(* IEC 61131-3 sources: mect_apps/Examples/Allarme_TPAC1007_04_AC/plc, 3 files *)

(* ---- Crosstable.gvl ---- *)
VAR_GLOBAL
	SetPoint_temp AT %QD0.4:REAL;
	Start AT %IX0.8.0:BOOL;
	Average_AnInp1 AT %QD0.776:REAL;
	Alarm_temp AT %IX0.780.0:BOOL;	(* Temperature alarm - Analog input 1 *)
	RTU0_TYPE_PORT AT %ID0.20000:UDINT;
	RTU0_BAUDRATE AT %ID0.20004:UDINT;
	RTU0_STATUS AT %ID0.20008:UDINT;
	RTU0_READS AT %ID0.20012:UDINT;
	RTU0_WRITES AT %ID0.20016:UDINT;
	RTU0_TIMEOUTS AT %ID0.20020:UDINT;
	RTU0_COMM_ERRORS AT %ID0.20024:UDINT;
	RTU0_LAST_ERROR AT %ID0.20028:UDINT;
	RTU0_WRITE_QUEUE AT %ID0.20032:UDINT;
	RTU0_READ_QUEUE AT %ID0.20036:UDINT;
	RTU1_TYPE_PORT AT %ID0.20040:UDINT;
	RTU1_BAUDRATE AT %ID0.20044:UDINT;
	RTU1_STATUS AT %ID0.20048:UDINT;
	RTU1_READS AT %ID0.20052:UDINT;
	RTU1_WRITES AT %ID0.20056:UDINT;
	RTU1_TIMEOUTS AT %ID0.20060:UDINT;
	RTU1_COMM_ERRORS AT %ID0.20064:UDINT;
	RTU1_LAST_ERROR AT %ID0.20068:UDINT;
	RTU1_WRITE_QUEUE AT %ID0.20072:UDINT;
	RTU1_READ_QUEUE AT %ID0.20076:UDINT;
	RTU3_TYPE_PORT AT %ID0.20080:UDINT;
	RTU3_BAUDRATE AT %ID0.20084:UDINT;
	RTU3_STATUS AT %ID0.20088:UDINT;
	RTU3_READS AT %ID0.20092:UDINT;
	RTU3_WRITES AT %ID0.20096:UDINT;
	RTU3_TIMEOUTS AT %ID0.20100:UDINT;
	RTU3_COMM_ERRORS AT %ID0.20104:UDINT;
	RTU3_LAST_ERROR AT %ID0.20108:UDINT;
	RTU3_WRITE_QUEUE AT %ID0.20112:UDINT;
	RTU3_READ_QUEUE AT %ID0.20116:UDINT;
	CAN0_TYPE_PORT AT %ID0.20120:UDINT;
	CAN0_BAUDRATE AT %ID0.20124:UDINT;
	CAN0_STATUS AT %ID0.20128:UDINT;
	CAN0_READS AT %ID0.20132:UDINT;
	CAN0_WRITES AT %ID0.20136:UDINT;
	CAN0_TIMEOUTS AT %ID0.20140:UDINT;
	CAN0_COMM_ERRORS AT %ID0.20144:UDINT;
	CAN0_LAST_ERROR AT %ID0.20148:UDINT;
	CAN0_WRITE_QUEUE AT %ID0.20152:UDINT;
	CAN0_READ_QUEUE AT %ID0.20156:UDINT;
	CAN1_TYPE_PORT AT %ID0.20160:UDINT;
	CAN1_BAUDRATE AT %ID0.20164:UDINT;
	CAN1_STATUS AT %ID0.20168:UDINT;
	CAN1_READS AT %ID0.20172:UDINT;
	CAN1_WRITES AT %ID0.20176:UDINT;
	CAN1_TIMEOUTS AT %ID0.20180:UDINT;
	CAN1_COMM_ERRORS AT %ID0.20184:UDINT;
	CAN1_LAST_ERROR AT %ID0.20188:UDINT;
	CAN1_WRITE_QUEUE AT %ID0.20192:UDINT;
	CAN1_READ_QUEUE AT %ID0.20196:UDINT;
	TCPS_TYPE_PORT AT %ID0.20200:UDINT;
	TCPS_IP_ADDRESS AT %ID0.20204:UDINT;
	TCPS_STATUS AT %ID0.20208:UDINT;
	TCPS_READS AT %ID0.20212:UDINT;
	TCPS_WRITES AT %ID0.20216:UDINT;
	TCPS_TIMEOUTS AT %ID0.20220:UDINT;
	TCPS_COMM_ERRORS AT %ID0.20224:UDINT;
	TCPS_LAST_ERROR AT %ID0.20228:UDINT;
	TCPS_WRITE_QUEUE AT %ID0.20232:UDINT;
	TCPS_READ_QUEUE AT %ID0.20236:UDINT;
	TCP0_TYPE_PORT AT %ID0.20240:UDINT;
	TCP0_IP_ADDRESS AT %ID0.20244:UDINT;
	TCP0_STATUS AT %ID0.20248:UDINT;
	TCP0_READS AT %ID0.20252:UDINT;
	TCP0_WRITES AT %ID0.20256:UDINT;
	TCP0_TIMEOUTS AT %ID0.20260:UDINT;
	TCP0_COMM_ERRORS AT %ID0.20264:UDINT;
	TCP0_LAST_ERROR AT %ID0.20268:UDINT;
	TCP0_WRITE_QUEUE AT %ID0.20272:UDINT;
	TCP0_READ_QUEUE AT %ID0.20276:UDINT;
	TCP1_TYPE_PORT AT %ID0.20280:UDINT;
	TCP1_IP_ADDRESS AT %ID0.20284:UDINT;
	TCP1_STATUS AT %ID0.20288:UDINT;
	TCP1_READS AT %ID0.20292:UDINT;
	TCP1_WRITES AT %ID0.20296:UDINT;
	TCP1_TIMEOUTS AT %ID0.20300:UDINT;
	TCP1_COMM_ERRORS AT %ID0.20304:UDINT;
	TCP1_LAST_ERROR AT %ID0.20308:UDINT;
	TCP1_WRITE_QUEUE AT %ID0.20312:UDINT;
	TCP1_READ_QUEUE AT %ID0.20316:UDINT;
	TCP2_TYPE_PORT AT %ID0.20320:UDINT;
	TCP2_IP_ADDRESS AT %ID0.20324:UDINT;
	TCP2_STATUS AT %ID0.20328:UDINT;
	TCP2_READS AT %ID0.20332:UDINT;
	TCP2_WRITES AT %ID0.20336:UDINT;
	TCP2_TIMEOUTS AT %ID0.20340:UDINT;
	TCP2_COMM_ERRORS AT %ID0.20344:UDINT;
	TCP2_LAST_ERROR AT %ID0.20348:UDINT;
	TCP2_WRITE_QUEUE AT %ID0.20352:UDINT;
	TCP2_READ_QUEUE AT %ID0.20356:UDINT;
	TCP3_TYPE_PORT AT %ID0.20360:UDINT;
	TCP3_IP_ADDRESS AT %ID0.20364:UDINT;
	TCP3_STATUS AT %ID0.20368:UDINT;
	TCP3_READS AT %ID0.20372:UDINT;
	TCP3_WRITES AT %ID0.20376:UDINT;
	TCP3_TIMEOUTS AT %ID0.20380:UDINT;
	TCP3_COMM_ERRORS AT %ID0.20384:UDINT;
	TCP3_LAST_ERROR AT %ID0.20388:UDINT;
	TCP3_WRITE_QUEUE AT %ID0.20392:UDINT;
	TCP3_READ_QUEUE AT %ID0.20396:UDINT;
	TCP4_TYPE_PORT AT %ID0.20400:UDINT;
	TCP4_IP_ADDRESS AT %ID0.20404:UDINT;
	TCP4_STATUS AT %ID0.20408:UDINT;
	TCP4_READS AT %ID0.20412:UDINT;
	TCP4_WRITES AT %ID0.20416:UDINT;
	TCP4_TIMEOUTS AT %ID0.20420:UDINT;
	TCP4_COMM_ERRORS AT %ID0.20424:UDINT;
	TCP4_LAST_ERROR AT %ID0.20428:UDINT;
	TCP4_WRITE_QUEUE AT %ID0.20432:UDINT;
	TCP4_READ_QUEUE AT %ID0.20436:UDINT;
	TCP5_TYPE_PORT AT %ID0.20440:UDINT;
	TCP5_IP_ADDRESS AT %ID0.20444:UDINT;
	TCP5_STATUS AT %ID0.20448:UDINT;
	TCP5_READS AT %ID0.20452:UDINT;
	TCP5_WRITES AT %ID0.20456:UDINT;
	TCP5_TIMEOUTS AT %ID0.20460:UDINT;
	TCP5_COMM_ERRORS AT %ID0.20464:UDINT;
	TCP5_LAST_ERROR AT %ID0.20468:UDINT;
	TCP5_WRITE_QUEUE AT %ID0.20472:UDINT;
	TCP5_READ_QUEUE AT %ID0.20476:UDINT;
	TCP6_TYPE_PORT AT %ID0.20480:UDINT;
	TCP6_IP_ADDRESS AT %ID0.20484:UDINT;
	TCP6_STATUS AT %ID0.20488:UDINT;
	TCP6_READS AT %ID0.20492:UDINT;
	TCP6_WRITES AT %ID0.20496:UDINT;
	TCP6_TIMEOUTS AT %ID0.20500:UDINT;
	TCP6_COMM_ERRORS AT %ID0.20504:UDINT;
	TCP6_LAST_ERROR AT %ID0.20508:UDINT;
	TCP6_WRITE_QUEUE AT %ID0.20512:UDINT;
	TCP6_READ_QUEUE AT %ID0.20516:UDINT;
	TCP7_TYPE_PORT AT %ID0.20520:UDINT;
	TCP7_IP_ADDRESS AT %ID0.20524:UDINT;
	TCP7_STATUS AT %ID0.20528:UDINT;
	TCP7_READS AT %ID0.20532:UDINT;
	TCP7_WRITES AT %ID0.20536:UDINT;
	TCP7_TIMEOUTS AT %ID0.20540:UDINT;
	TCP7_COMM_ERRORS AT %ID0.20544:UDINT;
	TCP7_LAST_ERROR AT %ID0.20548:UDINT;
	TCP7_WRITE_QUEUE AT %ID0.20552:UDINT;
	TCP7_READ_QUEUE AT %ID0.20556:UDINT;
	TCP8_TYPE_PORT AT %ID0.20560:UDINT;
	TCP8_IP_ADDRESS AT %ID0.20564:UDINT;
	TCP8_STATUS AT %ID0.20568:UDINT;
	TCP8_READS AT %ID0.20572:UDINT;
	TCP8_WRITES AT %ID0.20576:UDINT;
	TCP8_TIMEOUTS AT %ID0.20580:UDINT;
	TCP8_COMM_ERRORS AT %ID0.20584:UDINT;
	TCP8_LAST_ERROR AT %ID0.20588:UDINT;
	TCP8_WRITE_QUEUE AT %ID0.20592:UDINT;
	TCP8_READ_QUEUE AT %ID0.20596:UDINT;
	TCP9_TYPE_PORT AT %ID0.20600:UDINT;
	TCP9_IP_ADDRESS AT %ID0.20604:UDINT;
	TCP9_STATUS AT %ID0.20608:UDINT;
	TCP9_READS AT %ID0.20612:UDINT;
	TCP9_WRITES AT %ID0.20616:UDINT;
	TCP9_TIMEOUTS AT %ID0.20620:UDINT;
	TCP9_COMM_ERRORS AT %ID0.20624:UDINT;
	TCP9_LAST_ERROR AT %ID0.20628:UDINT;
	TCP9_WRITE_QUEUE AT %ID0.20632:UDINT;
	TCP9_READ_QUEUE AT %ID0.20636:UDINT;
	NODE_01_DEV_NODE AT %ID0.20688:UDINT;
	NODE_01_STATUS AT %ID0.20692:UDINT;
	NODE_02_DEV_NODE AT %ID0.20696:UDINT;
	NODE_02_STATUS AT %ID0.20700:UDINT;
	NODE_03_DEV_NODE AT %ID0.20704:UDINT;
	NODE_03_STATUS AT %ID0.20708:UDINT;
	NODE_04_DEV_NODE AT %ID0.20712:UDINT;
	NODE_04_STATUS AT %ID0.20716:UDINT;
	NODE_05_DEV_NODE AT %ID0.20720:UDINT;
	NODE_05_STATUS AT %ID0.20724:UDINT;
	NODE_06_DEV_NODE AT %ID0.20728:UDINT;
	NODE_06_STATUS AT %ID0.20732:UDINT;
	NODE_07_DEV_NODE AT %ID0.20736:UDINT;
	NODE_07_STATUS AT %ID0.20740:UDINT;
	NODE_08_DEV_NODE AT %ID0.20744:UDINT;
	NODE_08_STATUS AT %ID0.20748:UDINT;
	NODE_09_DEV_NODE AT %ID0.20752:UDINT;
	NODE_09_STATUS AT %ID0.20756:UDINT;
	NODE_10_DEV_NODE AT %ID0.20760:UDINT;
	NODE_10_STATUS AT %ID0.20764:UDINT;
	NODE_11_DEV_NODE AT %ID0.20768:UDINT;
	NODE_11_STATUS AT %ID0.20772:UDINT;
	NODE_12_DEV_NODE AT %ID0.20776:UDINT;
	NODE_12_STATUS AT %ID0.20780:UDINT;
	NODE_13_DEV_NODE AT %ID0.20784:UDINT;
	NODE_13_STATUS AT %ID0.20788:UDINT;
	NODE_14_DEV_NODE AT %ID0.20792:UDINT;
	NODE_14_STATUS AT %ID0.20796:UDINT;
	NODE_15_DEV_NODE AT %ID0.20800:UDINT;
	NODE_15_STATUS AT %ID0.20804:UDINT;
	NODE_16_DEV_NODE AT %ID0.20808:UDINT;
	NODE_16_STATUS AT %ID0.20812:UDINT;
	PLC_FWrevision AT %IW0.21200:UINT;	(* Firmware version *)
	PLC_HWconfig AT %IW0.21204:UINT;	(* Hardware configuration *)
	PLC_DigDir_1 AT %QX0.21208.0:BOOL;	(* Digital 1 direction (input = 0 output = 1) *)
	PLC_DigDir_2 AT %QX0.21212.0:BOOL;	(* Digital 2 direction (input = 0 output = 1) *)
	PLC_DigDir_3 AT %QX0.21216.0:BOOL;	(* Digital 3 direction (input = 0 output = 1) *)
	PLC_DigDir_4 AT %QX0.21220.0:BOOL;	(* Digital 4 direction (input = 0 output = 1) *)
	PLC_DigDir_5 AT %QX0.21224.0:BOOL;	(* Digital 5 direction (input = 0 output = 1) *)
	PLC_DigDir_6 AT %QX0.21228.0:BOOL;	(* Digital 6 direction (input = 0 output = 1) *)
	PLC_DigDir_7 AT %QX0.21232.0:BOOL;	(* Digital 7 direction (input = 0 output = 1) *)
	PLC_DigDir_8 AT %QX0.21236.0:BOOL;	(* Digital 8 direction (input = 0 output = 1) *)
	PLC_AnInConf_1 AT %QW0.21240:UINT;	(* Analog input 1 configuration *)
	PLC_AnInConf_2 AT %QW0.21244:UINT;	(* Analog input 2 configuration *)
	PLC_AnOutConf_1 AT %QW0.21248:UINT;	(* Analog output 1 configuration *)
	PLC_Reserved_1 AT %QW0.21252:UINT;	(* Reserved *)
	PLC_Reserved_2 AT %QW0.21256:UINT;	(* Reserved *)
	PLC_Reserved_3 AT %QW0.21260:UINT;	(* Reserved *)
	PLC_DigIn_1 AT %IX0.21264.0:BOOL;	(* Digital input 1 value *)
	PLC_DigIn_2 AT %IX0.21268.0:BOOL;	(* Digital input 2 value *)
	PLC_DigIn_3 AT %IX0.21272.0:BOOL;	(* Digital input 3 value *)
	PLC_DigIn_4 AT %IX0.21276.0:BOOL;	(* Digital input 4 value *)
	PLC_DigIn_5 AT %IX0.21280.0:BOOL;	(* Digital input 5 value *)
	PLC_DigIn_6 AT %IX0.21284.0:BOOL;	(* Digital input 6 value *)
	PLC_DigIn_7 AT %IX0.21288.0:BOOL;	(* Digital input 7 value *)
	PLC_DigIn_8 AT %IX0.21292.0:BOOL;	(* Digital input 8 value *)
	PLC_DigIn_9 AT %IX0.21296.0:BOOL;	(* Digital input 9 value *)
	PLC_DigIn_10 AT %IX0.21300.0:BOOL;	(* Digital input 10 value *)
	PLC_DigIn_11 AT %IX0.21304.0:BOOL;	(* Digital input 11 value *)
	PLC_DigIn_12 AT %IX0.21308.0:BOOL;	(* Digital input 12 value *)
	PLC_AnIn_1 AT %IW0.21312:INT;	(* Analog input 1 value *)
	PLC_AnIn_2 AT %IW0.21316:INT;	(* Analog input 2 value *)
	PLC_Reserved_4 AT %IW0.21320:INT;	(* Reserved *)
	PLC_Reserved_5 AT %IW0.21324:INT;	(* Reserved *)
	PLC_Reserved_6 AT %IW0.21328:INT;	(* Reserved *)
	PLC_Tamb AT %IW0.21332:INT;	(* Cold junction compensation value *)
	PLC_Encoder AT %ID0.21336:DINT;	(* Encoder reading value *)
	PLC_Capture AT %ID0.21340:UDINT;	(* Time between 2 input edges *)
	PLC_DigOut_1 AT %QX0.21344.0:BOOL;	(* Digital output 1 value *)
	PLC_DigOut_2 AT %QX0.21348.0:BOOL;	(* Digital output 2 value *)
	PLC_DigOut_3 AT %QX0.21352.0:BOOL;	(* Digital output 3 value *)
	PLC_DigOut_4 AT %QX0.21356.0:BOOL;	(* Digital output 4 value *)
	PLC_DigOut_5 AT %QX0.21360.0:BOOL;	(* Digital output 5 value *)
	PLC_DigOut_6 AT %QX0.21364.0:BOOL;	(* Digital output 6 value *)
	PLC_DigOut_7 AT %QX0.21368.0:BOOL;	(* Digital output 7 value *)
	PLC_DigOut_8 AT %QX0.21372.0:BOOL;	(* Digital output 8 value *)
	PLC_AnOut_1 AT %QW0.21376:INT;	(* Analog output 1 value *)
	PLC_Reserved_7 AT %QW0.21380:INT;	(* Reserved *)
	PLC_Reserved_8 AT %QW0.21384:INT;	(* Reserved *)
	PLC_Reserved_9 AT %QW0.21388:INT;	(* Reserved *)
	PLC_EncoderStart AT %QW0.21392:UINT;	(* Encoder - counter enable *)
	PLC_EncoderReset AT %QW0.21396:UINT;	(* Encoder reset *)
	PLC_Heartbeat AT %IW0.21400:UINT;	(* In - Out board function check *)
	PLC_StatusReg AT %IW0.21404:UINT;	(* In - Out board status *)
	PLC_AnIn1Filter AT %QW0.21408:UINT;	(* Analog input 1 filter *)
	PLC_AnIn2Filter AT %QW0.21412:UINT;	(* Analog input 2 filter *)
	PLC_time AT %ID0.21560:REAL;	(* Seconds since boot (reset each 24h) *)
	PLC_timeMin AT %ID0.21564:REAL;	(* 10 seconds window start *)
	PLC_timeMax AT %ID0.21568:REAL;	(* 10 seconds window stop *)
	PLC_timeWin AT %QD0.21572:REAL;	(* Graph display window *)
	PLC_Version AT %IW0.21576:UINT;	(* Run Time version *)
	PLC_EngineStatus AT %IW0.21580:UINT;	(* PLC status *)
	PLC_ResetValues AT %QX0.21584.0:BOOL;	(* Diagnostic variables reset *)
	PLC_buzzerOn AT %QX0.21588.0:BOOL;	(* Buzzer sound (enable = 1 disable = 0) *)
	PLC_PLC_Version AT %QW0.21592:UINT;	(* PLC application version *)
	PLC_HMI_Version AT %QW0.21596:UINT;	(* HMI application version *)
	PLC_Year AT %IW0.21640:UINT;	(* Currently year *)
	PLC_Month AT %IW0.21644:UINT;	(* Currently month *)
	PLC_Day AT %IW0.21648:UINT;	(* Currently day *)
	PLC_Hours AT %IW0.21652:UINT;	(* Currently hour *)
	PLC_Minutes AT %IW0.21656:UINT;	(* Currently minutes *)
	PLC_Seconds AT %IW0.21660:UINT;	(* Currently seconds *)
	PLC_UPTIME_s AT %ID0.21664:UDINT;	(* Uptime in seconds (wraps in 136 years) *)
	PLC_UPTIME_cs AT %ID0.21668:UDINT;	(* Uptime in centiseconds = 10 ms (wraps in 497 days) *)
	PLC_WATCHDOGEN AT %QX0.21672.0:BOOL;	(* Enable Watchdog *)
	PLC_WATCHDOG_ms AT %QD0.21676:UDINT;	(* Reset Watchdog timer *)
	PLC_PRODUCT_ID AT %ID0.21680:UDINT;	(* TP/TPAC/TPLC Product ID (Hex) *)
	PLC_SERIAL_NUMBER AT %ID0.21684:UDINT;	(* TP/TPAC/TPLC Serial Number *)
	PLC_HMI_PAGE AT %QD0.21688:DINT;	(* HMI Page (page100=0x00000100) *)
	PLC_BEEP_VOLUME AT %QB0.21740:BYTE;	(* Beep volume (when buzzerOn) *)
	PLC_TOUCH_VOLUME AT %QB0.21744:BYTE;	(* Touch volume *)
	PLC_ALARM_VOLUME AT %QB0.21748:BYTE;	(* Alarm volume (when alarm) *)
	PLC_BUZZER AT %QD0.21752:UDINT;	(* Enable dynamic buzzer sound (0x44332211 up=0x11(%) on=0x22(cs) off=0x33(cs) rep=0x44(times)) *)
END_VAR

(* ---- Init.st ---- *)
(*[[
]]*)
PROGRAM Init
#import "Crosstable.gvl"
#import "Resource1.gvl"
VAR

END_VAR

 	 PLC_AnInConf_1:= 7;     (* Analog inputs configuration : 0 = not configurated, 1 = current,
			                     2 =  voltage, 3 = TCJ, 4 = TCK,  5 = TCT, 6 = PT100E (NO decimal point),
							     7 = PT100R (decimal point), 8 = TCS, 9 = TCB, 10 = TCR	*)
     PLC_DigDir_2 := 1;      (* Digital I/O configuration: 0 = input, 1 = output*)
  	 PLC_AnOutConf_1 := 2;   (* Analog outputs configuration: 0 = not configurated, 1 = current, 2 = voltage, 3 = PWM *)
	 PLC_AnIn1Filter := 64;  (* a filter is used to stabilize the signal on analogue input 1 (PLC_AnIn1), it is a power of 2 number (64 = 2^8)*)

	 SetPoint_temp := 100.0; (* default set point *)
END_PROGRAM

(* ---- Normal.st ---- *)
(*[[
]]*)
PROGRAM Normal (*An alarm example. Esempio di allarme*)
#import "Crosstable.gvl"
#import "Resource1.gvl"
VAR

END_VAR
	(*See LADDER_ALARM program for ladder language / Vedere il programma LADDER_ALARM per il linguaggio ladder*)

     (*EN: Press "Start" to enable digital output 2 (PLC_DigOut_2) and voltage output of analog output 1 will be 6 V (PLC_AnOut_1 set as voltage, see "Init" program in the Task0_Init).
		   The variable "Average_AnInp1" contains the average of 10 PLC_AnIn_1 set as PT100 (temperature measurement) samples.
		   In the Crosstable (HMI) is set up an alarm (Alarm_temp): if "Average_AnInp1" is bigger than "SetPoint_temp"  value,  there will be an alarm.
		   When an alarm happens,  "Alarm_temp" is true and all the outputs will be disabled.
		   When "Start" is not pushed, all the outputs are disabled.

	   IT:Quando il bottone "Start" viene premuto si abilita l'uscita digitale 2 (PLC_DigOut_2) e l'uscita analogica 1 genera 6 V (PLC_AnOut_1 configurata
	   	  in tensione, vedere programma "Init" presente nel Task0_Init).
	      La variabile "Average_AnInp1" contiene la media mobile di 10 campioni dell'ingresso analogico 1 (PLC_AnIn_1 configurata in PT100).
		  Nella Crosstable (HMI) si è configurato un allarme (Alarm_temp): se "Average_AnInp1" è maggiore del valore di soglia "SetPoint_temp" si ha un allarme.
		  In caso di allarme si ha la variabile "Alarm_temp" uguale a true. In questo caso si disabiliteranno tutte le uscite.
		  Quando il buttone start non è premuto si hanno tutte le uscite disabilitate.*)

	  Average_AnInp1 := AVERAGE((INT_TO_REAL(PLC_AnIn_1) / 10.0), Average_AnInp1,10.0);  (*EN:AVERAGE is a function stored in ATCM_Common library (you need to download it into the project). IT: AVERAGE è una funzione presente nella libreria ATCM_Common (occorre importarla nel progetto)*)
	 if Start then
      	if Alarm_temp then
            PLC_DigOut_2 := false;(*alarm*)
	   		PLC_AnOut_1 := 0;
		else
			PLC_DigOut_2 := true; (*no alarm*)
	   		PLC_AnOut_1 := 600;
		end_if;
	  else
       	PLC_DigOut_2 := false;
	    PLC_AnOut_1 := 0;
 	  end_if;

END_PROGRAM
